% RSLogix 500 project I2P Job 11 - Andrew_Hoemmen.RSS, saved by version 10.00.00.00 %
PROJECT "ML03A"    % processor: Bul.1763 MicroLogix 1100 Series B %

PROGRAM FILES
  LAD 2   7 rungs

DATA FILES
  O0 OUTPUT  4 elements
  I1 INPUT  6 elements
  S2 STATUS  66 elements
  B3 BINARY  1 elements
  T4 TIMER  1 elements
  C5 COUNTER  1 elements
  R6 CONTROL  1 elements
  N7 INTEGER  1 elements
  F8 FLOAT  1 elements

LADDER 2
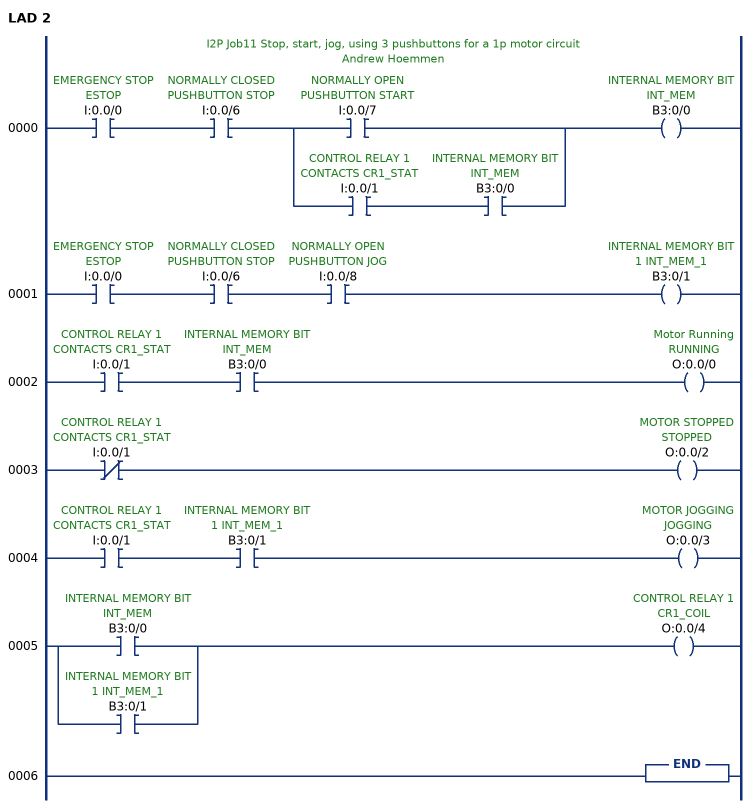
% Rung: 0 %
% I2P Job11 Stop, start, jog, using 3 pushbuttons for a 1p motor circuit
% Andrew Hoemmen %
SOR XIC I:0.0/0 XIC I:0.0/6 BST XIC I:0.0/7 NXB XIC I:0.0/1 XIC B3:0/0 BND OTE B3:0/0 EOR
%   I:0.0/0  ESTOP  "EMERGENCY STOP" %
%   I:0.0/6  STOP  "NORMALLY CLOSED PUSHBUTTON" %
%   I:0.0/7  START  "NORMALLY OPEN PUSHBUTTON" %
%   I:0.0/1  CR1_STAT  "CONTROL RELAY 1 CONTACTS" %
%   B3:0/0  INT_MEM  "INTERNAL MEMORY BIT" %
% Rung: 1 %
SOR XIC I:0.0/0 XIC I:0.0/6 XIC I:0.0/8 OTE B3:0/1 EOR
%   I:0.0/0  ESTOP  "EMERGENCY STOP" %
%   I:0.0/6  STOP  "NORMALLY CLOSED PUSHBUTTON" %
%   I:0.0/8  JOG  "NORMALLY OPEN PUSHBUTTON" %
%   B3:0/1  INT_MEM_1  "INTERNAL MEMORY BIT 1" %
% Rung: 2 %
SOR XIC I:0.0/1 XIC B3:0/0 OTE O:0.0/0 EOR
%   I:0.0/1  CR1_STAT  "CONTROL RELAY 1 CONTACTS" %
%   B3:0/0  INT_MEM  "INTERNAL MEMORY BIT" %
%   O:0.0/0  RUNNING  "Motor Running" %
% Rung: 3 %
SOR XIO I:0.0/1 OTE O:0.0/2 EOR
%   I:0.0/1  CR1_STAT  "CONTROL RELAY 1 CONTACTS" %
%   O:0.0/2  STOPPED  "MOTOR STOPPED" %
% Rung: 4 %
SOR XIC I:0.0/1 XIC B3:0/1 OTE O:0.0/3 EOR
%   I:0.0/1  CR1_STAT  "CONTROL RELAY 1 CONTACTS" %
%   B3:0/1  INT_MEM_1  "INTERNAL MEMORY BIT 1" %
%   O:0.0/3  JOGGING  "MOTOR JOGGING" %
% Rung: 5 %
SOR BST XIC B3:0/0 NXB XIC B3:0/1 BND OTE O:0.0/4 EOR
%   B3:0/0  INT_MEM  "INTERNAL MEMORY BIT" %
%   B3:0/1  INT_MEM_1  "INTERNAL MEMORY BIT 1" %
%   O:0.0/4  CR1_COIL  "CONTROL RELAY 1" %
% Rung: 6 %
SOR END EOR

OTHER DOCUMENTED ADDRESSES
  I:0.0/2  CR2_STATS  "CONTROL RELAY 2 CONTACTS"
  I:0.0/3  3PSS_A  "THREE POSITION SELECTOR SWITCH A POSITION"
  I:0.0/4  3PSS_B  "THREE POSITION SELECTOR SWITCH B POSITION"
  I:0.0/5  RUN_JOG  "TWO POSITION SELECTOR SWITCH"
  O:0.0/1  YEL_LT  "YELLOW LIGHT"
  O:0.0/5  CR2  "CONTROL RELAY 2"
